TYPE ST_RequestChangeState :
STRUCT
END_STRUCT
END_TYPE

(* stored: Version 1.1.0.1
   DUT ST_RequestChangeState: Id {c58c2240-9093-04af-02a3-8cca733321df} *)
